PROGRAM PRG_IM1K1_PPM
VAR
    {attribute 'pytmc' := '
        pv: IM1K1:PPM
        io: io
    '}
    {attribute 'TcLinkTo' := '.fbGige.iIlluminatorINT := TIIB[IM1K1-EL4004]^AO Outputs Channel 1^Analog output;
                              .fbGige.bGigePower := TIIB[IM1K1-EL2004]^Channel 2^Output;
                              .fbPowerMeter.iVoltageINT := TIIB[IM1K1-EL3062]^AI Standard Channel 1^Value;
                              .fbPowerMeter.fbThermoCouple.bError := TIIB[IM1K1-EL3314]^TC Inputs Channel 1^Status^Error;
                              .fbPowerMeter.fbThermoCouple.bUnderrange := TIIB[IM1K1-EL3314]^TC Inputs Channel 1^Status^Underrange;
                              .fbPowerMeter.fbThermoCouple.bOverrange := TIIB[IM1K1-EL3314]^TC Inputs Channel 1^Status^Overrange;
                              .fbPowerMeter.fbThermoCouple.iRaw := TIIB[IM1K1-EL3314]^TC Inputs Channel 1^Value;
                              .fbYagThermoCouple.bError := TIIB[IM1K1-EL3314]^TC Inputs Channel 2^Status^Error;
                              .fbYagThermoCouple.bUnderrange := TIIB[IM1K1-EL3314]^TC Inputs Channel 2^Status^Underrange;
                              .fbYagThermoCouple.bOverrange := TIIB[IM1K1-EL3314]^TC Inputs Channel 2^Status^Overrange;
                              .fbYagThermoCouple.iRaw := TIIB[IM1K1-EL3314]^TC Inputs Channel 2^Value'}
    fbIM1K1: FB_PPM;
END_VAR

fbIM1K1(
    stYStage := Main.M1,
    fPolished := -71.92,
    fFrosted := -97.93, // Actually a second polished yag
    fPower := -47.92,
    fOut := -8.82);

END_PROGRAM

(* stored: Version 1.1.0.1, ProductVersion 3.1.4022.18
   POU PRG_IM1K1_PPM: Id {d989df75-3cd2-4b27-b4dc-fd1dd338b294}, SpecialFunc None *)
